// TwinCAT 3 PLC project Cell_PLC
// Title: RoboFS Standard
// Company: HDS Global
// ProjectVersion: 1.0
// ProgramVersion: 3.1.4022.3
// libraries:
//   Controls Standard, * (Purav Dagli)
//   Tc2_DataExchange, * (Beckhoff Automation GmbH)
//   Tc2_MC2, * (Beckhoff Automation GmbH)
//   Tc2_Standard, * (Beckhoff Automation GmbH)
//   Tc2_System, * (Beckhoff Automation GmbH)
//   Tc2_Utilities, * (Beckhoff Automation GmbH)
//   Tc3_Module, * (Beckhoff Automation GmbH)
// project tree:
//   Cell/ Cell_Devices.TcPOU, Cell_SafetyMapping.TcPOU, Cell.TcGVL, Cell_Main.TcPOU, Cell_Sequencer.TcPOU
//   Cell/Comp01_UpperLvl/ Comp01.TcGVL, Comp01_Main.TcPOU, Comp01_Devices.TcPOU, Comp01_Sequencer.TcPOU
//   Cell/Comp02_LowerLvl/ Comp02_Devices.TcPOU, Comp02_Sequencer.TcPOU, Comp02.TcGVL, Comp02_Main.TcPOU
//   Cell/Interface/ Intfc_Left_PK.TcPOU, Intfc_Right_PK.TcPOU, Intfc.TcGVL, Intfc_Downstream_ML.TcPOU, Intfc_Upstream_ML.TcPOU
//   / PlcTask.TcTTO

CONFIGURATION Cell_PLC
    RESOURCE PLC ON TwinCAT3
        TASK PlcTask(INTERVAL := T#10ms, PRIORITY := 20);
        PROGRAM Cell_Main WITH PlcTask : Cell_Main;
        PROGRAM Intfc_Upstream_ML WITH PlcTask : Intfc_Upstream_ML;
        PROGRAM Intfc_Downstream_ML WITH PlcTask : Intfc_Downstream_ML;
        PROGRAM Intfc_Left_PK WITH PlcTask : Intfc_Left_PK;
        PROGRAM Intfc_Right_PK WITH PlcTask : Intfc_Right_PK;
    END_RESOURCE
END_CONFIGURATION

// ---- Cell/Comp01_UpperLvl/Comp01.TcGVL
{attribute 'qualified_only'}
VAR_GLOBAL
	StateManager			: StateManager;	
	D02_ACT1 				: Device_Actuator;
	D01_ACT2				: Device_Actuator;
	
	PartLoader_Pusher 				: Device_Servo;
	PartLoader_Pusher_Axis 			: Axis_Ref;
	
	D07_SRV2 				: Device_Servo;
	D07_SRV2_Axis 			: Axis_Ref;
END_VAR

VAR_GLOBAL PERSISTENT
	D06_SRV1_Moves 		: ARRAY [1..100] OF ServoMove;
	D07_SRV2_Moves 		: ARRAY [1..100] OF ServoMove;
END_VAR

// ---- Cell/Comp02_LowerLvl/Comp02.TcGVL
{attribute 'qualified_only'}
VAR_GLOBAL
	StateManager 	: StateManager;
END_VAR

// ---- Cell/Cell.TcGVL
{attribute 'qualified_only'}
VAR_GLOBAL
	StateManager : StateManager;
	iJogFwdButton  : BOOL;	
	iJogRevButton  : BOOL;	
	oJogButtonLight AT %Q* : BOOL;
	oSafetyReset AT %Q* : BOOL;
		iEStopOK AT %I* : BOOL;
END_VAR

// ---- Cell/Interface/Intfc.TcGVL
{attribute 'qualified_only'}
VAR_GLOBAL PERSISTENT
	Upstream_LaneA_Receiver	 		: Intfc_Receiver;
	Upstream_LaneB_Sender			: Intfc_Sender;
	Upstream_ExitLane_Sender		: Intfc_Sender;

	Downstream_LaneA_Sender			: Intfc_Sender;
	Downstream_LaneB_Receiver		: Intfc_Receiver;
	Downstream_ExitLane_Receiver	: Intfc_Receiver;
	
	LeftPick_Ingress_Sender			: Intfc_Sender;
	LeftPick_Egress_Receiver		: Intfc_Receiver;
	
	RightPick_Ingress_Sender		: Intfc_Sender;
	RightPick_Egress_Receiver		: Intfc_Receiver;
END_VAR

// ---- Cell/Cell_Main.TcPOU
PROGRAM Cell_Main
VAR_INPUT
	
END_VAR

VAR_OUTPUT

END_VAR

Cell.StateManager();
Cell_Sequencer();
Comp01_Main();

END_PROGRAM

// ---- Cell/Cell_Sequencer.TcPOU
PROGRAM Cell_Sequencer
VAR
END_VAR

CASE Cell.StateManager.oState OF
	State.Aborting:		Cell_SeqAborting();
	State.Aborted:		Cell_SeqAborted();
	State.Resetting:	Cell_SeqResetting();
	State.Stopped:		Cell_SeqStopped();
	State.Starting:		Cell_SeqStarting();
	State.Running:		Cell_SeqRunning();
	State.Pausing:		Cell_SeqPausing();
	State.Paused:		Cell_SeqPaused();
	State.Resuming:		Cell_SeqResuming();
	State.Stopping:		Cell_SeqStopping();	
END_CASE

ACTION Cell_SeqAborted:

END_ACTION

ACTION Cell_SeqAborting:
Comp01.StateManager.iCmd := Cmd.Abort;
//Comp02.StateManager.iCmd := Cmd.Abort;

IF Comp01.StateManager.oState = State.Aborted THEN //AND Comp02.StateManager.oState = State.Aborted THEN
	Cell.StateManager.iSeqComplete := TRUE;
END_IF
END_ACTION

ACTION Cell_SeqPaused:

END_ACTION

ACTION Cell_SeqPausing:
Comp01.StateManager.iCmd := Cmd.Pause;
//Comp02.StateManager.iCmd := Cmd.Pause;

IF Comp01.StateManager.oState = State.Paused THEN //AND Comp02.StateManager.oState = State.Paused THEN
	Cell.StateManager.iSeqComplete := TRUE;
END_IF
END_ACTION

ACTION Cell_SeqResetting:
Comp01.StateManager.iCmd := Cmd.Reset;
//Comp02.StateManager.iCmd := Cmd.Reset;

IF Comp01.StateManager.oState = State.Stopped THEN //AND Comp02.StateManager.oState = State.Stopped THEN
	Cell.StateManager.iSeqComplete := TRUE;
END_IF
END_ACTION

ACTION Cell_SeqResuming:
Comp01.StateManager.iCmd := Cmd.Resume;
//Comp02.StateManager.iCmd := Cmd.Resume;

IF Comp01.StateManager.oState = State.Running THEN //AND Comp02.StateManager.oState = State.Running THEN
	Cell.StateManager.iSeqComplete := TRUE;
END_IF
END_ACTION

ACTION Cell_SeqRunning:


IF Comp01.StateManager.oState = State.Stopping THEN //AND Comp02.StateManager.oState = State.Stopping THEN
	Cell.StateManager.iSeqComplete := TRUE;
END_IF
END_ACTION

ACTION Cell_SeqStarting:
Comp01.StateManager.iCmd := Cmd.Start;
//Comp02.StateManager.iCmd := Cmd.Start;

IF Comp01.StateManager.oState = State.Running THEN //AND Comp02.StateManager.oState = State.Running THEN
	Cell.StateManager.iSeqComplete := TRUE;
END_IF
END_ACTION

ACTION Cell_SeqStopped:

END_ACTION

ACTION Cell_SeqStopping:
Comp01.StateManager.iCmd := Cmd.Stop;
//Comp02.StateManager.iCmd := Cmd.Stop;

IF Comp01.StateManager.oState = State.Stopped THEN //AND Comp02.StateManager.oState = State.Stopped THEN
	Cell.StateManager.iSeqComplete := TRUE;
END_IF
END_ACTION

END_PROGRAM

// ---- Cell/Comp01_UpperLvl/Comp01_Main.TcPOU
PROGRAM Comp01_Main

Comp01.StateManager ();
Comp01_Sequencer();
Comp01_Devices();

IF Intfc.Upstream_LaneA_Receiver.iHandshake.WaitingToSend THEN
	Intfc.Upstream_LaneA_Receiver.oHandshake.ReadyToReceive := TRUE;
END_IF

END_PROGRAM

// ---- Cell/Comp01_UpperLvl/Comp01_Sequencer.TcPOU
PROGRAM Comp01_Sequencer
VAR
	ActiveStep 	: INT;
	Step1000	: Step;
	Step1010	: Step;
	Step1020	: Step;
	Step1030	: Step;
	Step1040	: Step;
	Step1050	: Step;
	Step1060	: Step;
	Step1070	: Step;
	Step1080	: Step;
	Step1090	: Step;
END_VAR

CASE Comp01.StateManager.oState OF
	State.Aborting:		Comp01_SeqAborting();
	State.Aborted:		Comp01_SeqAborted();
	State.Resetting:	Comp01_SeqResetting();
	State.Stopped:		Comp01_SeqStopped();
	State.Starting:		Comp01_SeqStarting();
	State.Running:		Comp01_SeqRunning();
	State.Pausing:		Comp01_SeqPausing();
	State.Paused:		Comp01_SeqPaused();
	State.Resuming:		Comp01_SeqResuming();
	State.Stopping:		
						Comp01_SeqRunning();
						Comp01_SeqStopping();	
END_CASE

ACTION Comp01_SeqAborted:

END_ACTION

ACTION Comp01_SeqAborting:
Comp01.PartLoader_Pusher.iCmd := CmdServo.Stop;
Comp01.D07_SRV2.iCmd := CmdServo.Stop;
IF Comp01.PartLoader_Pusher.oState = StateServo.Stopped AND Comp01.D07_SRV2.oState = StateServo.Stopped THEN
Comp01.StateManager.iSeqComplete := 1;
END_IF
END_ACTION

ACTION Comp01_SeqPaused:

END_ACTION

ACTION Comp01_SeqPausing:
Comp01.PartLoader_Pusher.iCmd := CmdServo.Stop;
Comp01.D07_SRV2.iCmd := CmdServo.Stop;
IF Comp01.PartLoader_Pusher.oState = StateServo.Stopped AND Comp01.D07_SRV2.oState = StateServo.Stopped THEN
Comp01.StateManager.iSeqComplete := 1;
END_IF
END_ACTION

ACTION Comp01_SeqResetting:
Comp01.StateManager.iSeqComplete := 1;
END_ACTION

ACTION Comp01_SeqResuming:
Comp01.StateManager.iSeqComplete := 1;
END_ACTION

ACTION Comp01_SeqRunning:
Step1000(	cDescription		:= 'Enable D06 Servo 1',
			cThisStep			:= 1000,
			cNextStep			:= 1010,
			cRecoveryStep		:= 1001,
			cTimeoutPreset 		:= T#5S,
			ioActiveStep 		:= ActiveStep);

IF Step1000.sActive THEN
			//Actions
			Comp01.PartLoader_Pusher.iCmd	:= CmdServo.Enable;
			
			//Completion Conditions
			IF Comp01.PartLoader_Pusher.oState = StateServo.Enabled OR Comp01.PartLoader_Pusher.oState = StateServo.Stopped THEN
			Step1000.iComplete	:= TRUE;
			END_IF
END_IF			

//=============================================================================//
			
Step1010(	cDescription	:= 'Start D06 Servo 1 Move 1',
			cThisStep		:= 1010,
			cNextStep		:= 1020,
			cRecoveryStep	:= 1011,
			cTimeoutPreset 	:= T#5S,
			ioActiveStep 	:= ActiveStep);

IF Step1010.sActive THEN
			//Actions
			Comp01.PartLoader_Pusher.iMoveIndex := 1;
			Comp01.PartLoader_Pusher.iCmd	:= CmdServo.StartMove;
			
			//Completion Conditions
			IF Comp01.PartLoader_Pusher.oState = StateServo.MoveInProgress THEN
			Step1010.iComplete	:= TRUE;
			END_IF
END_IF		

//=============================================================================//

Step1020(	cDescription	:= 'Wait for D06 Servo 1 Move 1 Complete',
			cThisStep		:= 1020,
			cNextStep		:= 1030,
			cRecoveryStep	:= 1021,
			cTimeoutPreset 	:= T#5S,
			ioActiveStep 	:= ActiveStep);

IF Step1020.sActive THEN
			//Actions
			
			//Completion Conditions
			IF Comp01.PartLoader_Pusher.oState = StateServo.MoveComplete AND Comp01.PartLoader_Pusher.sMoveIndex = Comp01.PartLoader_Pusher.iMoveIndex THEN
			Step1020.iComplete	:= TRUE;
			END_IF
END_IF		

//=============================================================================//
			
Step1030(	cDescription	:= 'Extend D01 Actuator 1',
			cThisStep		:= 1030,
			cNextStep		:= 1040,
			cRecoveryStep	:= 1031,
			cTimeoutPreset 	:= T#5S,
			ioActiveStep 	:= ActiveStep);

IF Step1030.sActive THEN
			//Actions
			//Comp01.D01_ACT1.iCmd	:= CmdActuator.Extend;
			
			//Completion Conditions
			IF Comp01.D02_ACT1.oState = StateActuator.Extended THEN
			Step1030.iComplete	:= TRUE;
			END_IF
END_IF		

//=============================================================================//

Step1040(	cDescription	:= 'Start D06 Servo 1 Move 2',
			cThisStep		:= 1040,
			cNextStep		:= 1050,
			cRecoveryStep	:= 1041,
			cTimeoutPreset 	:= T#5S,
			ioActiveStep 	:= ActiveStep);

IF Step1040.sActive THEN
			//Actions
			Comp01.PartLoader_Pusher.iMoveIndex := 2;
			Comp01.PartLoader_Pusher.iCmd	:= CmdServo.StartMove;
			
			//Completion Conditions
			IF Comp01.PartLoader_Pusher.oState = StateServo.MoveComplete AND Comp01.PartLoader_Pusher.sMoveIndex = Comp01.PartLoader_Pusher.iMoveIndex THEN
			Step1040.iComplete	:= TRUE;
			END_IF
END_IF		

//=============================================================================//


Step1050(	cDescription	:= 'Wait for D06 Servo 1 Move 2 Complete',
			cThisStep		:= 1050,
			cNextStep		:= 1060,
			cRecoveryStep	:= 1051,
			cTimeoutPreset 	:= T#5S,
			ioActiveStep 	:= ActiveStep);

IF Step1050.sActive THEN
			//Actions
			
			//Completion Conditions
			IF Comp01.PartLoader_Pusher.oState = StateServo.MoveComplete AND Comp01.PartLoader_Pusher.sMoveIndex = Comp01.PartLoader_Pusher.iMoveIndex THEN
			Step1050.iComplete	:= TRUE;
			END_IF
END_IF		

//=============================================================================//
			
Step1060(	cDescription	:= 'Retract D01 Actuator 1',
			cThisStep		:= 1060,
			cNextStep		:= 1070,
			cRecoveryStep	:= 1061,
			cTimeoutPreset 	:= T#5S,
			ioActiveStep 	:= ActiveStep);

IF Step1060.sActive THEN
			//Actions
			Comp01.D02_ACT1.iCmd	:= CmdActuator.Retract;
			
			//Completion Conditions
			IF Comp01.D02_ACT1.oState = StateActuator.Retracted THEN
			Step1060.iComplete	:= TRUE;
			END_IF
END_IF		

//=============================================================================//

Step1070(	cDescription	:= 'Disable D06 Servo 1',
			cThisStep		:= 1070,
			cNextStep		:= 1080,
			cRecoveryStep	:= 1071,
			cTimeoutPreset 	:= T#5S,
			ioActiveStep 	:= ActiveStep);

IF Step1070.sActive THEN
			//Actions
			Comp01.PartLoader_Pusher.iCmd := CmdServo.Disable;
			
			//Completion Conditions
			IF Comp01.PartLoader_Pusher.oState = StateServo.Disabled THEN
			Step1070.iComplete	:= TRUE;
			Comp01.StateManager.iSeqComplete := TRUE;
			END_IF
END_IF		

//=============================================================================//
END_ACTION

ACTION Comp01_SeqStarting:
Comp01.StateManager.iSeqComplete := 1;
END_ACTION

ACTION Comp01_SeqStopped:

END_ACTION

ACTION Comp01_SeqStopping:

END_ACTION

END_PROGRAM

// ---- Cell/Comp01_UpperLvl/Comp01_Devices.TcPOU
PROGRAM Comp01_Devices
VAR
	Step_0: Step;
END_VAR

Lifts();
Servos();

ACTION Conveyors:
// NETWORK 1
END_ACTION

ACTION ConveyorStops:
// NETWORK 1
END_ACTION

ACTION LiftAndTransfers:
// NETWORK 1
END_ACTION

ACTION Lifts:
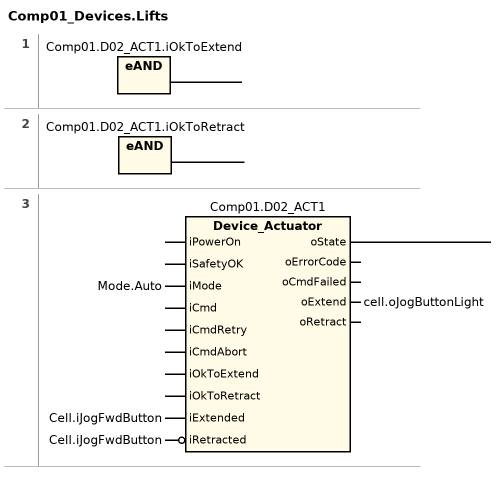
// NETWORK 1
Comp01.D02_ACT1.iOkToExtend(); // eAND

// NETWORK 2
Comp01.D02_ACT1.iOkToRetract(); // eAND

// NETWORK 3
Comp01.D02_ACT1(
    iMode := Mode.Auto,
    iExtended := Cell.iJogFwdButton,
    iRetracted := NOT Cell.iJogFwdButton,
    oExtend => cell.oJogButtonLight); // Device_Actuator
END_ACTION

ACTION Servos:
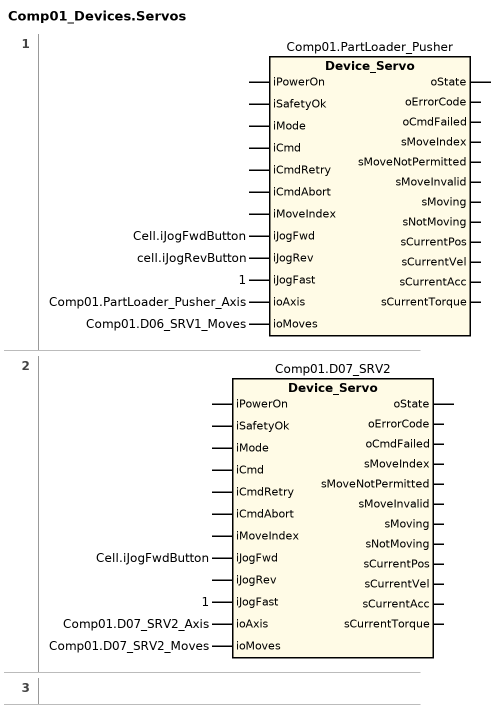
// NETWORK 1
Comp01.PartLoader_Pusher(
    iJogFwd := Cell.iJogFwdButton,
    iJogRev := cell.iJogRevButton,
    iJogFast := 1,
    ioAxis := Comp01.PartLoader_Pusher_Axis,
    ioMoves := Comp01.D06_SRV1_Moves); // Device_Servo

// NETWORK 2
Comp01.D07_SRV2(
    iJogFwd := Cell.iJogFwdButton,
    iJogFast := 1,
    ioAxis := Comp01.D07_SRV2_Axis,
    ioMoves := Comp01.D07_SRV2_Moves); // Device_Servo

// NETWORK 3
END_ACTION

END_PROGRAM

// ---- Cell/Interface/Intfc_Upstream_ML.TcPOU
PROGRAM Intfc_Upstream_ML
VAR
	Upstream_Upper_LaneA_Comm		: FB_ReadAdsSymByName;
	Upstream_Upper_LaneB_Comm		: FB_ReadAdsSymByName;
	Upstream_Upper_ExitLane_Comm	: FB_ReadAdsSymByName;
	Upstream_Lower_LaneA_Comm		: FB_ReadAdsSymByName;
	Upstream_Lower_LaneB_Comm		: FB_ReadAdsSymByName;
	Upstream_Lower_ExitLane_Comm	: FB_ReadAdsSymByName;
	UpdateRate						: TIME;
	UpdateTimer						: TON;
	UpdateCounter					: CTU;
END_VAR

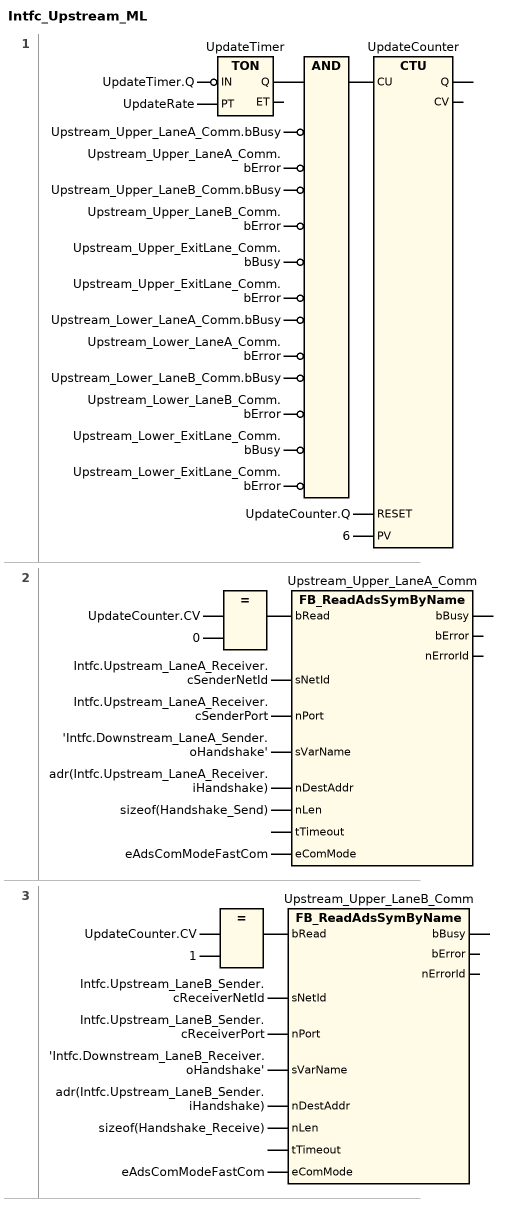
// NETWORK 1
UpdateTimer(IN := NOT UpdateTimer.Q, PT := UpdateRate); // TON
UpdateCounter(
    CU := UpdateTimer.Q AND NOT Upstream_Upper_LaneA_Comm.bBusy AND NOT Upstream_Upper_LaneA_Comm.bError AND NOT Upstream_Upper_LaneB_Comm.bBusy AND NOT Upstream_Upper_LaneB_Comm.bError AND NOT Upstream_Upper_ExitLane_Comm.bBusy AND NOT Upstream_Upper_ExitLane_Comm.bError AND NOT Upstream_Lower_LaneA_Comm.bBusy AND NOT Upstream_Lower_LaneA_Comm.bError AND NOT Upstream_Lower_LaneB_Comm.bBusy AND NOT Upstream_Lower_LaneB_Comm.bError AND NOT Upstream_Lower_ExitLane_Comm.bBusy AND NOT Upstream_Lower_ExitLane_Comm.bError,
    RESET := UpdateCounter.Q,
    PV := 6); // CTU

// NETWORK 2
Upstream_Upper_LaneA_Comm(
    bRead := UpdateCounter.CV = 0,
    sNetId := Intfc.Upstream_LaneA_Receiver.cSenderNetId,
    nPort := Intfc.Upstream_LaneA_Receiver.cSenderPort,
    sVarName := 'Intfc.Downstream_LaneA_Sender.oHandshake',
    nDestAddr := adr(Intfc.Upstream_LaneA_Receiver.iHandshake),
    nLen := sizeof(Handshake_Send),
    eComMode := eAdsComModeFastCom); // FB_ReadAdsSymByName

// NETWORK 3
Upstream_Upper_LaneB_Comm(
    bRead := UpdateCounter.CV = 1,
    sNetId := Intfc.Upstream_LaneB_Sender.cReceiverNetId,
    nPort := Intfc.Upstream_LaneB_Sender.cReceiverPort,
    sVarName := 'Intfc.Downstream_LaneB_Receiver.oHandshake',
    nDestAddr := adr(Intfc.Upstream_LaneB_Sender.iHandshake),
    nLen := sizeof(Handshake_Receive),
    eComMode := eAdsComModeFastCom); // FB_ReadAdsSymByName

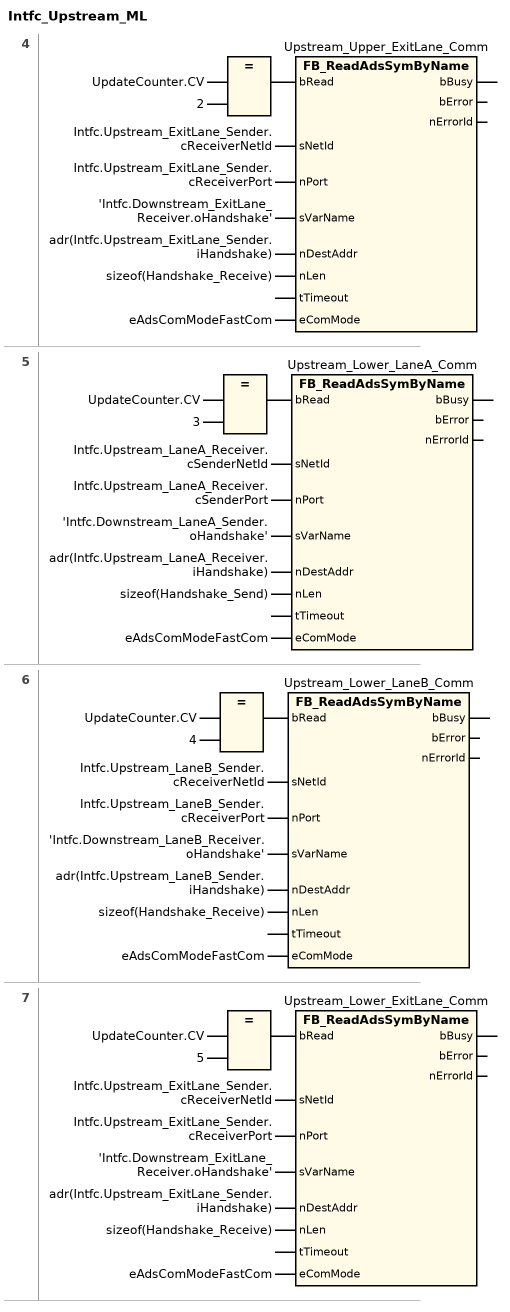
// NETWORK 4
Upstream_Upper_ExitLane_Comm(
    bRead := UpdateCounter.CV = 2,
    sNetId := Intfc.Upstream_ExitLane_Sender.cReceiverNetId,
    nPort := Intfc.Upstream_ExitLane_Sender.cReceiverPort,
    sVarName := 'Intfc.Downstream_ExitLane_Receiver.oHandshake',
    nDestAddr := adr(Intfc.Upstream_ExitLane_Sender.iHandshake),
    nLen := sizeof(Handshake_Receive),
    eComMode := eAdsComModeFastCom); // FB_ReadAdsSymByName

// NETWORK 5
Upstream_Lower_LaneA_Comm(
    bRead := UpdateCounter.CV = 3,
    sNetId := Intfc.Upstream_LaneA_Receiver.cSenderNetId,
    nPort := Intfc.Upstream_LaneA_Receiver.cSenderPort,
    sVarName := 'Intfc.Downstream_LaneA_Sender.oHandshake',
    nDestAddr := adr(Intfc.Upstream_LaneA_Receiver.iHandshake),
    nLen := sizeof(Handshake_Send),
    eComMode := eAdsComModeFastCom); // FB_ReadAdsSymByName

// NETWORK 6
Upstream_Lower_LaneB_Comm(
    bRead := UpdateCounter.CV = 4,
    sNetId := Intfc.Upstream_LaneB_Sender.cReceiverNetId,
    nPort := Intfc.Upstream_LaneB_Sender.cReceiverPort,
    sVarName := 'Intfc.Downstream_LaneB_Receiver.oHandshake',
    nDestAddr := adr(Intfc.Upstream_LaneB_Sender.iHandshake),
    nLen := sizeof(Handshake_Receive),
    eComMode := eAdsComModeFastCom); // FB_ReadAdsSymByName

// NETWORK 7
Upstream_Lower_ExitLane_Comm(
    bRead := UpdateCounter.CV = 5,
    sNetId := Intfc.Upstream_ExitLane_Sender.cReceiverNetId,
    nPort := Intfc.Upstream_ExitLane_Sender.cReceiverPort,
    sVarName := 'Intfc.Downstream_ExitLane_Receiver.oHandshake',
    nDestAddr := adr(Intfc.Upstream_ExitLane_Sender.iHandshake),
    nLen := sizeof(Handshake_Receive),
    eComMode := eAdsComModeFastCom); // FB_ReadAdsSymByName

END_PROGRAM

// ---- Cell/Interface/Intfc_Downstream_ML.TcPOU
PROGRAM Intfc_Downstream_ML
VAR
END_VAR

// NETWORK 1

END_PROGRAM

// ---- Cell/Interface/Intfc_Left_PK.TcPOU
PROGRAM Intfc_Left_PK
VAR
END_VAR

// NETWORK 1

END_PROGRAM

// ---- Cell/Interface/Intfc_Right_PK.TcPOU
PROGRAM Intfc_Right_PK
VAR
END_VAR

// NETWORK 1

END_PROGRAM

// ---- Cell/Cell_Devices.TcPOU
PROGRAM Cell_Devices
VAR
END_VAR

END_PROGRAM

// ---- Cell/Cell_SafetyMapping.TcPOU
PROGRAM Cell_SafetyMapping
VAR

END_VAR

END_PROGRAM

// ---- Cell/Comp02_LowerLvl/Comp02_Devices.TcPOU
PROGRAM Comp02_Devices
VAR
END_VAR

END_PROGRAM

// ---- Cell/Comp02_LowerLvl/Comp02_Sequencer.TcPOU
PROGRAM Comp02_Sequencer
VAR
	ActiveStep 	: INT;
	Step1000	: Step;
	Step1100	: Step;
END_VAR

CASE Comp02.StateManager.oState OF
	State.Aborting:		Comp02_SeqAborting();
	State.Aborted:		Comp02_SeqAborted();
	State.Resetting:	Comp02_SeqResetting();
	State.Stopped:		Comp02_SeqStopped();
	State.Starting:		Comp02_SeqStarting();
	State.Running:		Comp02_SeqRunning();
	State.Pausing:		Comp02_SeqPausing();
	State.Paused:		Comp02_SeqPaused();
	State.Resuming:		Comp02_SeqResuming();
	State.Stopping:		Comp02_SeqStopping();	
END_CASE

ACTION Comp02_SeqAborted:

END_ACTION

ACTION Comp02_SeqAborting:

END_ACTION

ACTION Comp02_SeqPaused:

END_ACTION

ACTION Comp02_SeqPausing:

END_ACTION

ACTION Comp02_SeqResetting:

END_ACTION

ACTION Comp02_SeqResuming:

END_ACTION

ACTION Comp02_SeqRunning:
Step1000(	cDescription		:= 'Raise Blade Stop',
			cThisStep			:= 1000,
			cNextStep			:= 1100,
			cRecoveryStep		:= 1050,
			cTimeoutPreset 		:= T#5S,
			ioActiveStep 		:= ActiveStep);

IF Step1000.sActive THEN
			Comp01.D02_ACT1.iCmd	:= CmdActuator.Extend;
			Step1000.iComplete	:= TRUE;
END_IF			

//=============================================================================//
			
Step1100(	cDescription	:= 'Enable D06 Servo 1',
			cThisStep		:= 1100,
			cNextStep		:= 1200,
			cRecoveryStep	:= 1150,
			cTimeoutPreset 	:= T#5S,
			ioActiveStep 	:= ActiveStep);

IF Step1100.sActive THEN
			Comp01.PartLoader_Pusher.iCmd	:= CmdServo.Enable;
			Step1100.iComplete	:= TRUE;
END_IF		

//=============================================================================//
END_ACTION

ACTION Comp02_SeqStarting:

END_ACTION

ACTION Comp02_SeqStopped:

END_ACTION

ACTION Comp02_SeqStopping:

END_ACTION

END_PROGRAM

// ---- Cell/Comp02_LowerLvl/Comp02_Main.TcPOU
PROGRAM Comp02_Main

END_PROGRAM
